INTERFACE VacuumController

METHOD GetCurrentPressure : REAL
END_METHOD

METHOD Run : BOOL
END_METHOD

METHOD SetPressureRequired : BOOL
VAR_INPUT
	Pressure : REAL;
END_VAR
END_METHOD

METHOD Stop : BOOL
END_METHOD

END_INTERFACE

(* stored: Version 1.1.0.1, ProductVersion 3.1.4022.16
   Itf VacuumController: Id {a6ba872a-680c-43c9-bbd3-617ff5b97c87}
   Method GetCurrentPressure: Id {b4b0a566-08c1-409c-9474-042f0a202c71}
   Method Run: Id {52599611-8733-4e90-8e2d-548edbbc782f}
   Method SetPressureRequired: Id {d5fda7c4-e0fa-4237-8451-ee7d4b8d7e1a}
   Method Stop: Id {325ea40d-0a1d-4adf-8d28-015b11c19d28} *)
